TYPE PiperStatus :
STRUCT
	state : MACHINE_STATE;
	subState : DINT;
END_STRUCT
END_TYPE

(* stored: Version 1.1.0.1, ProductVersion 3.1.4024.12
   DUT PiperStatus: Id {c45b24db-af61-4757-a3bf-0b74bf7fe770} *)
